{attribute 'GeneratedUsingTerminal: EK1100-0000-0018'}
{attribute addProperty BoxType "EK1100-0000-0018"}
{attribute addProperty Id "Beckhoff_EPP3xxxEK1122Beckhoff_EPP3xxxEK1122_6CDF68111480"}
{attribute addProperty CRC "3529204970"}
{attribute addProperty Size "1480"}
TYPE Beckhoff_EPP3xxx_D25B64EA EXTENDS EK1100_AB5A9467 :
STRUCT
	{attribute addProperty Name "Beckhoff_EPP3xxxEK1122"}
	Beckhoff_EPP3xxxEK1122 : Beckhoff_EPP3xxxEK1122_6CDF6811;
END_STRUCT
END_TYPE

(* stored: Version 1.2.0.0, ProductVersion 3.1.4024.9
   DUT Beckhoff_EPP3xxx_D25B64EA: Id {1d3e070c-48b7-427a-b8e7-ca71a96be67f} *)
